// TwinCAT 3 PLC project Sample03
// ProgramVersion: 3.1.4023.0
// libraries:
//   Tc2_Standard, * (Beckhoff Automation GmbH)
//   Tc2_System, * (Beckhoff Automation GmbH)
//   Tc3_Module, * (Beckhoff Automation GmbH)
// project tree:
//   / PlcTask.TcTTO
//   POUs/ ClassDiagram.TcCD (not stored), FB_ContractEmployee.TcPOU, FB_Employee.TcPOU, FB_FullTimeEmployee.TcPOU, I_Employee.TcIO, MAIN.TcPOU
// real-time tasks:
//   TASK PlcTask: cycle T#10ms, priority 20, ADS port 350

CONFIGURATION Sample03
    RESOURCE PLC ON TwinCAT3
        TASK PlcTask(INTERVAL := T#10ms, PRIORITY := 20);
        PROGRAM MAIN WITH PlcTask : MAIN;
    END_RESOURCE
END_CONFIGURATION

// ---- POUs/I_Employee.TcIO
INTERFACE I_Employee

METHOD GetFullName : STRING
VAR_INPUT
END_VAR
END_METHOD

METHOD GetMonthlySalary : LREAL
VAR_INPUT
END_VAR
END_METHOD

PROPERTY nPersonnelNumber : UINT
GET
END_GET
SET
END_SET
END_PROPERTY

PROPERTY sFirstName : STRING
GET
END_GET
SET
END_SET
END_PROPERTY

PROPERTY sLastName : STRING
GET
END_GET
SET
END_SET
END_PROPERTY

END_INTERFACE

// ---- POUs/MAIN.TcPOU
PROGRAM MAIN
VAR
	fbFullTimeEmployee	:	FB_FullTimeEmployee;
	fbContractEmployee	:	FB_ContractEmployee;
	refEmployee			:	REFERENCE TO FB_Employee;
	ipEmployee			:	I_Employee;	
	aFullName			:	ARRAY[1..2] OF STRING;
	aMonthlySalary		:	ARRAY[1..2] OF LREAL;
END_VAR

fbFullTimeEmployee.nPersonnelNumber := 1;
fbFullTimeEmployee.sFirstName := 'John';
fbFullTimeEmployee.sLastName := 'Taylor';
fbFullTimeEmployee.nAnnualSalary := 60000;
// access via concrete FB
aFullName[1] := fbFullTimeEmployee.GetFullName();
aMonthlySalary[1] := fbFullTimeEmployee.GetMonthlySalary();
// access via abstract FB
refEmployee REF= fbFullTimeEmployee;
aFullName[1] := refEmployee.GetFullName();
aMonthlySalary[1] := refEmployee.GetMonthlySalary();
// access via interface
ipEmployee := fbFullTimeEmployee;
aFullName[1] := ipEmployee.GetFullName();
aMonthlySalary[1] := ipEmployee.GetMonthlySalary();

fbContractEmployee.nPersonnelNumber := 2;
fbContractEmployee.sFirstName := 'Tim';
fbContractEmployee.sLastName := 'Brown';
fbContractEmployee.nMonthlyHours := 160;
fbContractEmployee.nHourlyPay := 35;
// access via concrete FB
aFullName[2] := fbContractEmployee.GetFullName();
aMonthlySalary[2] := fbContractEmployee.GetMonthlySalary();
// access via abstract FB
refEmployee REF= fbContractEmployee;
aFullName[2] := refEmployee.GetFullName();
aMonthlySalary[2] := refEmployee.GetMonthlySalary();
// access via interface
ipEmployee := fbContractEmployee;
aFullName[2] := ipEmployee.GetFullName();
aMonthlySalary[2] := ipEmployee.GetMonthlySalary();

END_PROGRAM

// ---- POUs/FB_FullTimeEmployee.TcPOU
{attribute 'hide_all_locals'}
FUNCTION_BLOCK PUBLIC FB_FullTimeEmployee EXTENDS FB_Employee
VAR_INPUT
END_VAR
VAR_OUTPUT
END_VAR
VAR
	nAnnualSalaryBacking	:	UINT;
END_VAR

METHOD PUBLIC GetMonthlySalary : LREAL
VAR_INPUT
END_VAR
GetMonthlySalary := nAnnualSalary / 12;
END_METHOD

{attribute 'monitoring' := 'variable'}
PROPERTY PUBLIC nAnnualSalary : UINT
GET
nAnnualSalary := nAnnualSalaryBacking;
END_GET
SET
nAnnualSalaryBacking := nAnnualSalary;
END_SET
END_PROPERTY

END_FUNCTION_BLOCK

// ---- POUs/FB_Employee.TcPOU
{attribute 'hide_all_locals'}
FUNCTION_BLOCK PUBLIC ABSTRACT FB_Employee IMPLEMENTS I_Employee
VAR_INPUT
END_VAR
VAR_OUTPUT
END_VAR
VAR
	nPersonnelNumberBacking :	UINT;
	sFirstNameBacking		:	STRING;
	sLastNameBacking		:	STRING;
END_VAR

METHOD PUBLIC GetFullName : STRING
VAR_INPUT
END_VAR
GetFullName := CONCAT(CONCAT(CONCAT(CONCAT(TO_STRING(nPersonnelNumber), ': '), sFirstName), ' '), sLastName);
END_METHOD

METHOD PUBLIC ABSTRACT GetMonthlySalary : LREAL
VAR_INPUT
END_VAR
END_METHOD

{attribute 'monitoring' := 'variable'}
PROPERTY PUBLIC nPersonnelNumber : UINT
GET
nPersonnelNumber := nPersonnelNumberBacking;
END_GET
SET
nPersonnelNumberBacking := nPersonnelNumber;
END_SET
END_PROPERTY

{attribute 'monitoring' := 'variable'}
PROPERTY PUBLIC sFirstName : STRING
GET
sFirstName := sFirstNameBacking;
END_GET
SET
sFirstNameBacking := sFirstName;
END_SET
END_PROPERTY

{attribute 'monitoring' := 'variable'}
PROPERTY PUBLIC sLastName : STRING
GET
sLastName := sLastNameBacking;
END_GET
SET
sLastNameBacking := sLastName;
END_SET
END_PROPERTY

END_FUNCTION_BLOCK

// ---- POUs/FB_ContractEmployee.TcPOU
{attribute 'hide_all_locals'}
FUNCTION_BLOCK PUBLIC FB_ContractEmployee EXTENDS FB_Employee
VAR_INPUT
END_VAR
VAR_OUTPUT
END_VAR
VAR
	nHourlyPayBacking		:	UINT;
	nMonthlyHoursBacking	:	UINT;
END_VAR

METHOD PUBLIC GetMonthlySalary : LREAL
VAR_INPUT
END_VAR
GetMonthlySalary := nMonthlyHours * nHourlyPay;
END_METHOD

{attribute 'monitoring' := 'variable'}
PROPERTY PUBLIC nHourlyPay : UINT
GET
nHourlyPay := nHourlyPayBacking;
END_GET
SET
nHourlyPayBacking := nHourlyPay;
END_SET
END_PROPERTY

{attribute 'monitoring' := 'variable'}
PROPERTY PUBLIC nMonthlyHours : UINT
GET
nMonthlyHours := nMonthlyHoursBacking;
END_GET
SET
nMonthlyHoursBacking := nMonthlyHours;
END_SET
END_PROPERTY

END_FUNCTION_BLOCK
